PROGRAM prgLynusVar
VAR
	fbVarInfo		: FB_VarInfo;
	fbRW1			: FB_ReadWrite;
	fbRW2			: FB_ReadWrite;
END_VAR

fbVarInfo(
	bReadInfo:= , 
	eTMCFile:= eSelectTMCFile.eDontUseTMCFile, 
	eSavePositionTMCFile:= eSavePositionOnPLC.ePostionC, 
	udiCounterFoundVariables=> , 
	bError=> , 
	bBusy=> , 
	byProgress=> , 
	udiErrorCodeOut=> , 
	eErrorVarInfo_Out=> , 
	sVarWithError=> );
	
fbRW1();
fbRW2();

END_PROGRAM

(* stored: Version 1.1.0.1, ProductVersion 3.1.4024.9
   POU prgLynusVar: Id {f0d96063-d05f-4608-97c4-1a5b90627e8f}, SpecialFunc None *)
